FUNCTION INTERNAL _FindBestChunk : Result
VAR_INPUT
	nRequesterId		: UDINT;
    nRequestedSize     	: UDINT;
END_VAR
VAR_OUTPUT
    nNewId             	: UDINT;
    nNewSize            : UDINT;
END_VAR
VAR
	i					: UDINT;
	j					: UDINT;
END_VAR

// Loop through stEntry to find the best chunk
FOR i := 1 TO Param.BROADCAST_CAP DO
	IF _Broadcast.stEntry[i].iSignal <> 0 AND_THEN _Broadcast.stEntry[i].iSignal.id <> nRequesterId THEN
		// Skip over occupied blocks
		i := _Broadcast.stEntry[i].iSignal.id + _Broadcast.stEntry[i].iSignal.size - 1;
	ELSE
		// Start of a free chunk and measure its size
		FOR j := 0 TO Param.BROADCAST_CAP DO
			IF _Broadcast.stEntry[i + j].iSignal <> 0 AND_THEN _Broadcast.stEntry[i].iSignal.id <> nRequesterId THEN
				EXIT;
			ELSIF Param.BROADCAST_CAP <= i + j THEN
				EXIT;
			END_IF			
		END_FOR
		
		// If the chunk is smaller but still fits assign a new best fit
		IF nNewSize = 0 THEN
			nNewId := i;
			nNewSize := j + 1;
		ELSIF  nRequestedSize <= j + 1 AND_THEN nNewSize > j + 1 THEN
			nNewId := i;
			nNewSize := nRequestedSize;
		END_IF
		
		IF _Broadcast.stEntry[i + j].iSignal = 0 THEN
			i := i + j;
		ELSE
			i := i + j - 1;
		END_IF
		
	END_IF
END_FOR

IF nNewSize > 0 THEN
	nNewSize := nRequestedSize;
	_FindBestChunk := Ok;
ELSE
	_FindBestChunk := Error;
END_IF

END_FUNCTION

(* stored: Version 1.1.0.1
   POU _FindBestChunk: Id {1a257033-abe9-4a30-b199-a186888c3328}, SpecialFunc None *)
